//==================================================================================================
//								RJM Maszyny sp. z o.o.
//									04.02.2022
//	Elektrozawor 3 na 2
// 	v1.0	|| TC v 3.1.4024.22		|| - pierwsza wersja
//==================================================================================================
INTERFACE I_Elektrozawor_3na2

//==================================================================================================
//								RJM Maszyny sp. z o.o.
//									04.02.2022
//	Włączenie cewki - wyjscie 2
// 	v1.0	|| TC v 3.1.4024.22		|| - pierwsza wersja
//==================================================================================================
METHOD Wlacz
VAR_INPUT
END_VAR
END_METHOD

//==================================================================================================
//								RJM Maszyny sp. z o.o.
//									04.02.2022
//	Wyłączenie cewki - wyjscie 2
// 	v1.0	|| TC v 3.1.4024.22		|| - pierwsza wersja
//==================================================================================================
METHOD Wylacz
VAR_INPUT
END_VAR
END_METHOD

END_INTERFACE

(* stored: Version 1.1.0.1, ProductVersion 3.1.4024.11
   Itf I_Elektrozawor_3na2: Id {1a257659-20e8-4cb3-9ee3-6f60c1d28f89}
   Method Wlacz: Id {2c642abe-2eb9-413d-b8f8-b31439cb127e}
   Method Wylacz: Id {a2c79c79-124b-4071-91ab-664a0a4b2a9b} *)
